FUNCTION LimitRealNumber : REAL
VAR_INPUT
	IN : REAL;
	LowLimit : REAL;
	HighLimit : REAL;
END_VAR
VAR
END_VAR

LimitRealNumber:= IN;

IF (IN<LowLimit) THEN
	LimitRealNumber:= LowLimit;
END_IF

IF (IN>HighLimit) THEN
	LimitRealNumber:= HighLimit;
END_IF

END_FUNCTION

(* stored: Version 1.1.0.1, ProductVersion 3.1.4024.15
   POU LimitRealNumber: Id {226f105c-14a9-4992-bdc2-3523434d8ab9}, SpecialFunc None *)
